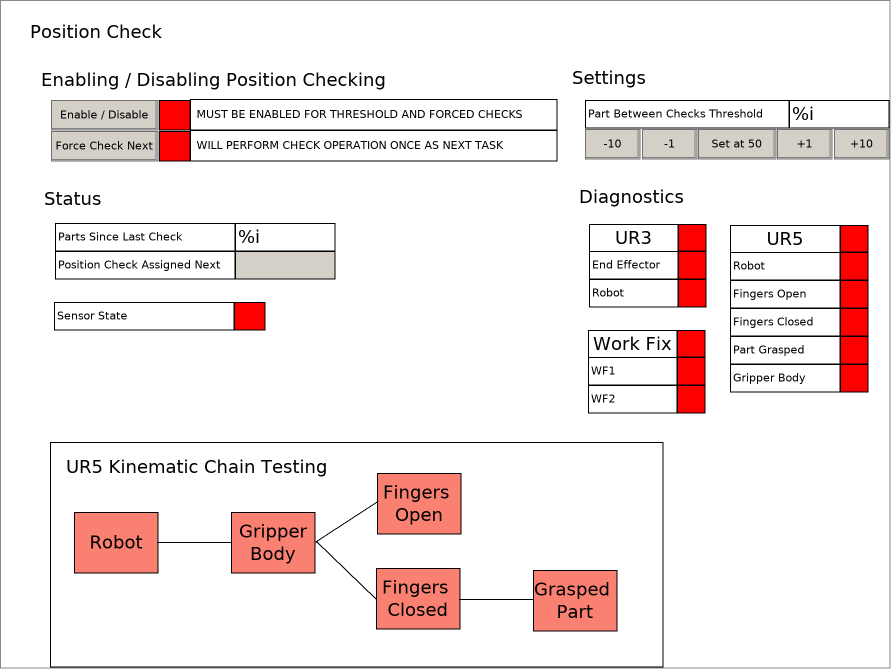
VISUALIZATION PositionCheck  // 891x669
    RoundedRectangle (50,442 613x225)
    Rectangle (55,223 180x28), "Parts Since Last Check"
    Rectangle (235,223 100x28), "%i", text variable: Global.nPartsSincePosCheck
    Rectangle (589,224 89x28), "UR3"
    Rectangle (589,251 89x28), "End Effector"
    Rectangle (589,279 89x28), "Robot"
    Rectangle (678,224 28x27), colour toggle: global.UR3PosCheck[1] and global.UR3PosCheck[2]
    Rectangle (678,279 28x28), colour toggle: Global.UR3PosCheck[2]
    Rectangle (678,251 28x28), colour toggle: Global.UR3PosCheck[1]
    Rectangle (730,225 110x28), "UR5"
    Rectangle (730,252 110x28), "Robot"
    Rectangle (730,280 110x28), "Fingers Open"
    Rectangle (840,225 28x27), colour toggle: Global.UR5PosCheck[1] and Global.UR5PosCheck[2] and Global.UR5PosCheck[3] and Global.UR5PosCheck[4] and Global.UR5PosCheck[5]
    Rectangle (840,280 28x28), colour toggle: Global.UR5PosCheck[3]
    Rectangle (840,252 28x28), colour toggle: Global.UR5PosCheck[5]
    Rectangle (588,330 89x28), "Work Fix"
    Rectangle (588,357 89x28), "WF1"
    Rectangle (588,385 89x28), "WF2"
    Rectangle (677,330 28x27)
    Rectangle (677,385 28x28)
    Rectangle (677,357 28x28)
    Rectangle (730,308 110x28), "Fingers Closed"
    Rectangle (840,308 28x28), colour toggle: Global.UR5PosCheck[2]
    Rectangle (730,336 110x28), "Part Grasped"
    Rectangle (840,336 28x28), colour toggle: Global.UR5PosCheck[1]
    Rectangle (730,364 110x28), "Gripper Body"
    Rectangle (840,364 28x28), colour toggle: Global.UR5PosCheck[4]
    Label (41,184 260x30), "Status"
    Button (51,100 107x30), "Enable / Disable"
        OnMouseClick: toggle Global.bEnablePosCheck
    Rectangle (159,100 31x30), colour toggle: Global.bEnablePosCheck
    Label (27,17 260x30), "Position Check"
    Rectangle (585,100 204x28), "Part Between Checks Threshold"
    Rectangle (789,100 100x28), "%i", text variable: Global.nPosCheckThreshold
    Button (51,131 107x30), "Force Check Next"
        OnMouseClick: toggle Global.bForcePosCheck
    Rectangle (159,131 31x30), colour toggle: Global.bForcePosCheck
    Rectangle (190,130 367x31), "WILL PERFORM CHECK OPERATION ONCE AS NEXT TASK"
    Rectangle (190,99 367x31), "MUST BE ENABLED FOR THRESHOLD AND FORCED CHECKS"
    Label (38,65 360x30), "Enabling / Disabling Position Checking"
    Label (569,63 260x30), "Settings"
    Button (698,129 78x30), "Set at 50"
        OnMouseClick: execute { Global.nPosCheckThreshold := 50; }
    Button (777,129 55x30), "+1"
        OnMouseClick: execute { Global.nPosCheckThreshold := Global.nPosCheckThreshold + 1; }
    Button (834,129 55x30), "+10"
        OnMouseClick: execute { Global.nPosCheckThreshold := Global.nPosCheckThreshold + 10; }
    Button (585,129 55x30), "-10"
        OnMouseClick: execute { Global.nPosCheckThreshold := Global.nPosCheckThreshold - 10; }
    Button (642,129 55x30), "-1"
        OnMouseClick: execute { Global.nPosCheckThreshold := Global.nPosCheckThreshold - 1; }
    Label (576,182 260x30), "Diagnostics"
    Rectangle (55,251 180x28), "Position Check Assigned Next"
    Rectangle (235,251 100x28), colour toggle: Global.bForcePosCheck
    Rectangle (54,302 180x28), "Sensor State"
    Rectangle (234,302 31x28), colour toggle: Global.bPosSensorState
    RoundedRectangle (74,512 84x61), "Robot", colour toggle: Global.UR5PosCheck[1]
    RoundedRectangle (231,512 84x61), "Gripper Body", colour toggle: Global.UR5PosCheck[2]
    RoundedRectangle (377,473 84x61), "Fingers Open", colour toggle: Global.UR5PosCheck[3]
    RoundedRectangle (376,568 84x61), "Fingers Closed", colour toggle: Global.UR5PosCheck[4]
    RoundedRectangle (533,570 84x61), "Grasped Part", colour toggle: Global.UR5PosCheck[5]
    Line (157,542) (231,542)
    Line (315,542) (378,501)
    Line (316,541) (376,599)
    Line (459,599) (533,599)
    Label (63,452 344x30), "UR5 Kinematic Chain Testing"
END_VISUALIZATION

(* stored: Version 1.1.0.1, ProductVersion 3.1.4020.12
   Visu PositionCheck: Id {3341829e-0435-4451-a885-3c81574f2bed} *)
